// Mitsubishi GX Works2 project: testrs485v2   PLC: FX3U/FX3UC

PROGRAM MAIN
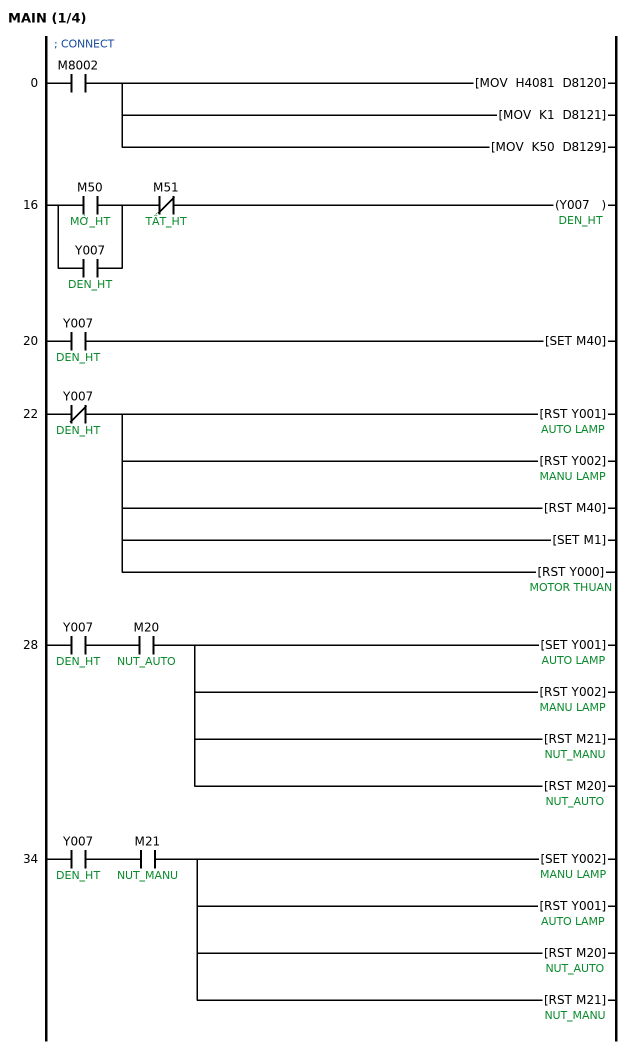
; CONNECT
0     LD      M8002
      MOV     H4081 D8120
      MOV     K1 D8121
      MOV     K50 D8129
16    LD      M50  ; MỞ_HT
      OR      Y007  ; DEN_HT
      ANI     M51  ; TẮT_HT
      OUT     Y007  ; DEN_HT
20    LD      Y007  ; DEN_HT
      SET     M40
22    LDI     Y007  ; DEN_HT
      RST     Y001  ; AUTO LAMP
      RST     Y002  ; MANU LAMP
      RST     M40
      SET     M1
      RST     Y000  ; MOTOR THUAN
28    LD      Y007  ; DEN_HT
      AND     M20  ; NUT_AUTO
      SET     Y001  ; AUTO LAMP
      RST     Y002  ; MANU LAMP
      RST     M21  ; NUT_MANU
      RST     M20  ; NUT_AUTO
34    LD      Y007  ; DEN_HT
      AND     M21  ; NUT_MANU
      SET     Y002  ; MANU LAMP
      RST     Y001  ; AUTO LAMP
      RST     M20  ; NUT_AUTO
      RST     M21  ; NUT_MANU
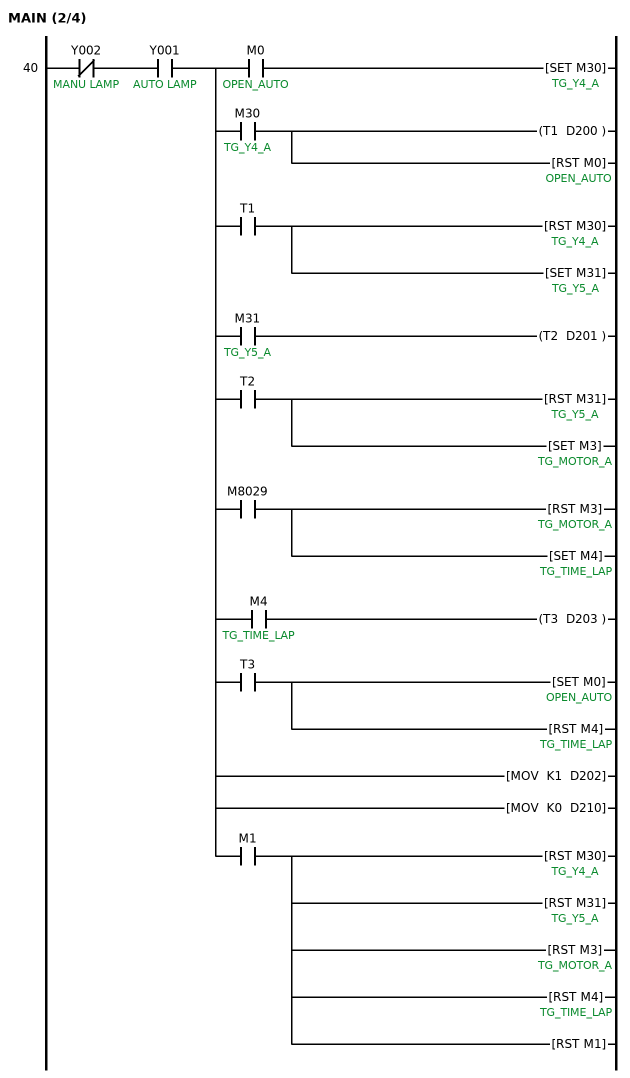
40    LDI     Y002  ; MANU LAMP
      AND     Y001  ; AUTO LAMP
      MPS
      AND     M0  ; OPEN_AUTO
      SET     M30  ; TG_Y4_A
      MRD
      AND     M30  ; TG_Y4_A
      OUT     T1 D200
      RST     M0  ; OPEN_AUTO
      MRD
      AND     T1
      RST     M30  ; TG_Y4_A
      SET     M31  ; TG_Y5_A
      MRD
      AND     M31  ; TG_Y5_A
      OUT     T2 D201
      MRD
      AND     T2
      RST     M31  ; TG_Y5_A
      SET     M3  ; TG_MOTOR_A
      MRD
      AND     M8029
      RST     M3  ; TG_MOTOR_A
      SET     M4  ; TG_TIME_LAP
      MRD
      AND     M4  ; TG_TIME_LAP
      OUT     T3 D203
      MRD
      AND     T3
      SET     M0  ; OPEN_AUTO
      RST     M4  ; TG_TIME_LAP
      MPP
      MOV     K1 D202
      MOV     K0 D210
      AND     M1
      RST     M30  ; TG_Y4_A
      RST     M31  ; TG_Y5_A
      RST     M3  ; TG_MOTOR_A
      RST     M4  ; TG_TIME_LAP
      RST     M1
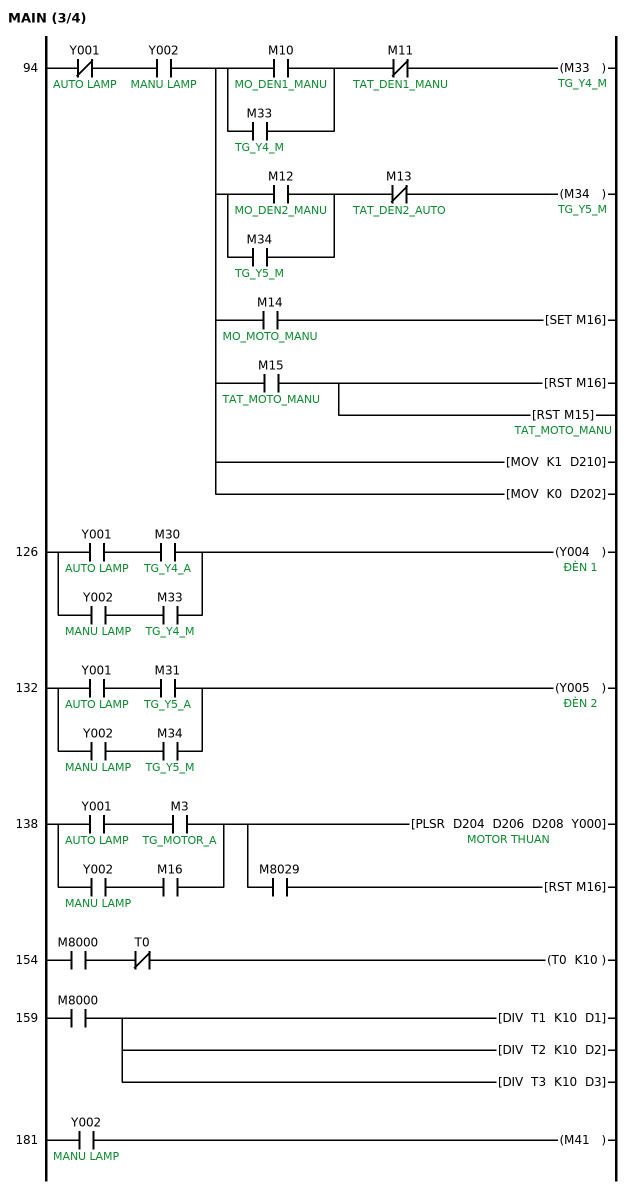
94    LDI     Y001  ; AUTO LAMP
      AND     Y002  ; MANU LAMP
      MPS
      LD      M10  ; MO_DEN1_MANU
      OR      M33  ; TG_Y4_M
      ANB
      ANI     M11  ; TAT_DEN1_MANU
      OUT     M33  ; TG_Y4_M
      MRD
      LD      M12  ; MO_DEN2_MANU
      OR      M34  ; TG_Y5_M
      ANB
      ANI     M13  ; TAT_DEN2_AUTO
      OUT     M34  ; TG_Y5_M
      MRD
      AND     M14  ; MO_MOTO_MANU
      SET     M16
      MRD
      AND     M15  ; TAT_MOTO_MANU
      RST     M16
      RST     M15  ; TAT_MOTO_MANU
      MPP
      MOV     K1 D210
      MOV     K0 D202
126   LD      Y001  ; AUTO LAMP
      AND     M30  ; TG_Y4_A
      LD      Y002  ; MANU LAMP
      AND     M33  ; TG_Y4_M
      ORB
      OUT     Y004  ; ĐÈN 1
132   LD      Y001  ; AUTO LAMP
      AND     M31  ; TG_Y5_A
      LD      Y002  ; MANU LAMP
      AND     M34  ; TG_Y5_M
      ORB
      OUT     Y005  ; ĐÈN 2
138   LD      Y001  ; AUTO LAMP
      AND     M3  ; TG_MOTOR_A
      LD      Y002  ; MANU LAMP
      AND     M16
      ORB
      PLSR    D204 D206 D208 Y000  ; MOTOR THUAN
      AND     M8029
      RST     M16
154   LD      M8000
      ANI     T0
      OUT     T0 K10
159   LD      M8000
      DIV     T1 K10 D1
      DIV     T2 K10 D2
      DIV     T3 K10 D3
181   LD      Y002  ; MANU LAMP
      OUT     M41
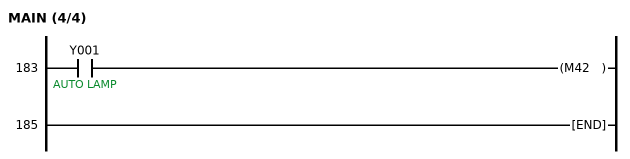
183   LD      Y001  ; AUTO LAMP
      OUT     M42
185   END
END_PROGRAM

// device comments not shown above
Y003  ; MOTO NGHICH
